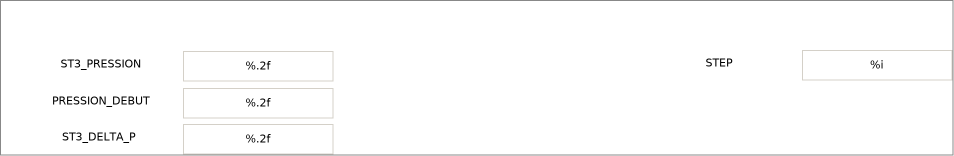
VISUALIZATION ST3  // 954x156
    Textfield (183,51 150x30), "%.2f", text variable: ST3_PRESSION
    Label (26,49 150x30), "ST3_PRESSION"
    Textfield (183,88 150x30), "%.2f", text variable: ST3_ETANCHEITE.PRESSION_DEBUT
    Label (26,86 150x30), "PRESSION_DEBUT"
    Textfield (183,124 150x30), "%.2f", text variable: ST3_DELTA_P
    Label (24,122 150x30), "ST3_DELTA_P"
    Label (644,48 150x30), "STEP"
    Textfield (802,50 150x30), "%i", text variable: IOs_Variables.PROG_STEPS.ST3
END_VISUALIZATION

(* stored: Version 1.1.0.1, ProductVersion 3.1.0.26
   Visu ST3: Id {2973a40d-293c-4812-a93d-80137f6f50e8} *)
